// TwinCAT 3 PLC project FirstCode
// ProgramVersion: 3.1.4023.0
// libraries:
//   Tc2_Standard, * (Beckhoff Automation GmbH)
//   Tc2_System, * (Beckhoff Automation GmbH)
//   Tc2_Utilities, * (Beckhoff Automation GmbH)
//   Tc3_Module, * (Beckhoff Automation GmbH)
// project tree:
//   DUTs/ E_EventType.TcDUT, ST_Event.TcDUT
//   / PlcTask.TcTTO
//   POUs/ EventLogger.TcPOU, MAIN.TcPOU, UpdateEventWithSystemTime.TcPOU
// real-time tasks:
//   TASK PlcTask: cycle T#10ms, priority 20, ADS port 350

CONFIGURATION FirstCode
    RESOURCE PLC ON TwinCAT3
        TASK PlcTask(INTERVAL := T#10ms, PRIORITY := 20);
        PROGRAM MAIN WITH PlcTask : MAIN;
    END_RESOURCE
END_CONFIGURATION

// ---- DUTs/E_EventType.TcDUT
{attribute 'qualified_only'}
{attribute 'strict'}
TYPE E_EventType :
(
	Alarm := 0,
	Message:= 1
);
END_TYPE

// ---- DUTs/ST_Event.TcDUT
TYPE ST_Event :
STRUCT
    eEventType: E_EventType;
	eEventSeverity: TcEventSeverity;
	nEventIdentity : UDINT;
	sEventText: STRING(255);
	dtTimeStamp: DATE_AND_TIME;
	
END_STRUCT
END_TYPE

// ---- POUs/MAIN.TcPOU
PROGRAM MAIN
VAR
	stThisIsFirstEvent: ST_Event;
	bBoolean: BOOL :=FALSE;
	
END_VAR

IF NOT bBoolean THEN
UpdateEventWithSystemTime(stEvent:= stThisIsFirstEvent);
bBoolean := TRUE;
END_IF

END_PROGRAM

// ---- POUs/UpdateEventWithSystemTime.TcPOU
FUNCTION UpdateEventWithSystemTime 
VAR_INPUT
	stEvent : REFERENCE TO ST_Event;
END_VAR
VAR
	fbGETSYSTEMTIME : GETSYSTEMTIME;
	stFileTime: T_FILETIME;
	
END_VAR

fbGETSYSTEMTIME( timeLoDW => stFileTime.dwLowDateTime,
	              timeHiDW => stFileTime.dwHighDateTime);


stEvent.dtTimestamp := FILETIME_TO_DT(fileTime := stFileTime);

END_FUNCTION

// ---- POUs/EventLogger.TcPOU
FUNCTION_BLOCK EventLogger
VAR_INPUT
END_VAR
VAR_OUTPUT
END_VAR
VAR
END_VAR

END_FUNCTION_BLOCK
